// TIA Portal V19 export
TYPE "C406_VAR_CAD_TYPIC"
   STRUCT
      POS_STS { ExternalAccessible := 'False'; ExternalVisible := 'False'; ExternalWritable := 'False'} : USInt;   // Stand van de calamiteitendoorsteek
      BST { ExternalAccessible := 'False'; ExternalVisible := 'False'; ExternalWritable := 'False'} : USInt;   // Bestuurbaarheid
   END_STRUCT;
END_TYPE
